TYPE TcaRackFeederService :
STRUCT

END_STRUCT
END_TYPE

(* stored: Version 1.1.0.1
   DUT TcaRackFeederService: Id {0b5824bf-617d-4872-9ca0-76829cbb8a88} *)
